RoboDK station: Pick and Place.rdk

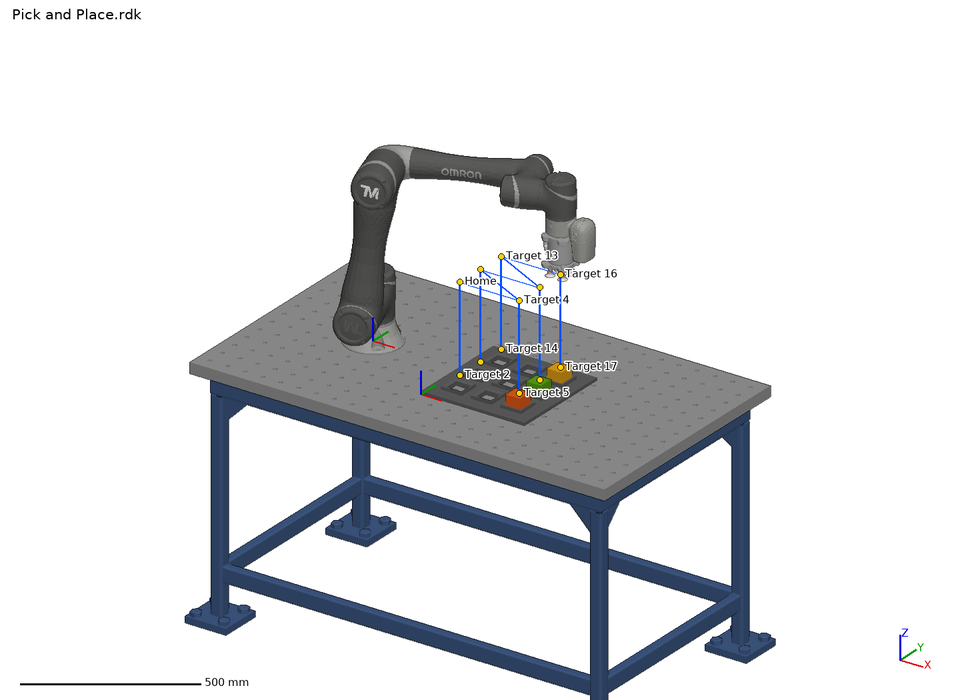
[picture v0: the station drawn from its stored meshes, robots at their saved joint values, targets as dots, program paths as lines]
Station Pick and Place (saved by RoboDK 5.9.2). Poses are relative to the parent item; angles as X-Y-Z fixed-axis rotations.
  - frame Omron TM5-900 Base at (0, 0, 0) mm
    - robot Omron TM5-900: 6 axes, payload 4 kg, reach 900 mm, repeatability 0.05 mm, weight 22.6 kg
        modified DH rows (alpha deg, a mm, theta deg, d mm): 0, 0, 0, 145.2; 90, 0, 90, 0; 0, 429, 0, 0; 0, 411, -90, 122.3; -90, 0, 0, 106.5; 90, 0, 180, 114.15
        joint limits [-270, -180, -155, -180, -180, -270] to [270, 180, 155, 180, 180, 270]; home [0, 0, 90, -90, 90, 0]; saved at [19.778, 6.994, 82.568, 0.438, 90, 19.778]
      - tool SMC ZXP7A01-ZP25C-X1 Vacuum Gripper, TCP at (0, 0, 125) mm, size 88 x 106.8 x 127.9 mm
  - object Table 1400x800x800mm at (0, 0, 0) mm, size 1420 x 820 x 800 mm, geometry from Table-1400x800x800mm.sld
  - frame Reference Frame at (300, -200, 0) mm
    - object Pallete  at (0, 0, 0) mm, size 350 x 350 x 20 mm, geometry from Pallete .step
    - target Home (Cartesian target) at (77.5, 77.7, 335.05) mm, rotated rx 180 ry 0 rz 90 deg; joints [0, -18.954, 105.709, 3.244, 90, 0] of Omron TM5-900
    - target Target 2 (Cartesian target) at (77.5, 77.7, 50) mm, rotated rx 180 ry 0 rz 90 deg; joints [0, -3.452, 137.214, -43.761, 90, 0] of Omron TM5-900
    - target Target 3 (Cartesian target) at (77.5, 77.7, 335) mm, rotated rx 180 ry 0 rz 90 deg; joints [0, -18.954, 105.717, 3.237, 90, 0] of Omron TM5-900
    - target Target 4 (Cartesian target) at (277.5, 77.7, 335) mm, rotated rx 180 ry 0 rz 90 deg; joints [0, 8.043, 81.376, 0.581, 90, 0] of Omron TM5-900
    - target Target 5 (Cartesian target) at (277.5, 77.7, 50) mm, rotated rx 180 ry 0 rz 90 deg; joints [0, 20.58, 108.244, -38.825, 90, 0] of Omron TM5-900
    - target Target 6 (Cartesian target) at (277.5, 77.7, 335) mm, rotated rx 180 ry 0 rz 90 deg; joints [0, 8.043, 81.376, 0.581, 90, 0] of Omron TM5-900
    - target Target 7 (Cartesian target) at (77.5, 177.7, 335) mm, rotated rx 180 ry 0 rz 90 deg; joints [15.489, -21.689, 107.458, 4.231, 90, 15.489] of Omron TM5-900
    - target Target 8 (Cartesian target) at (77.5, 177.7, 50) mm, rotated rx 180 ry 0 rz 90 deg; joints [15.489, -6.322, 139.731, -43.409, 90, 15.489] of Omron TM5-900
    - target Target 9 (Cartesian target) at (77.5, 177.7, 335) mm, rotated rx 180 ry 0 rz 90 deg; joints [15.489, -21.689, 107.458, 4.231, 90, 15.489] of Omron TM5-900
    - target Target 10 (Cartesian target) at (277.5, 177.7, 335) mm, rotated rx 180 ry 0 rz 90 deg; joints [10.006, 6.337, 83.305, 0.358, 90, 10.006] of Omron TM5-900
    - target Target 11 (Cartesian target) at (277.5, 177.7, 50) mm, rotated rx 180 ry 0 rz 90 deg; joints [10.006, 19.191, 110.269, -39.46, 90, 10.006] of Omron TM5-900
    - target Target 12 (Cartesian target) at (277.5, 177.7, 335) mm, rotated rx 180 ry 0 rz 90 deg; joints [10.006, 6.337, 83.305, 0.358, 90, 10.006] of Omron TM5-900
    - target Target 13 (Cartesian target) at (77.5, 277.7, 335) mm, rotated rx 180 ry 0 rz 90 deg; joints [30.132, -20.621, 106.794, 3.828, 90, 30.132] of Omron TM5-900
    - target Target 14 (Cartesian target) at (77.5, 277.7, 50) mm, rotated rx 180 ry 0 rz 90 deg; joints [30.132, -5.185, 138.759, -43.573, 90, 30.132] of Omron TM5-900
    - target Target 15 (Cartesian target) at (77.5, 277.7, 335) mm, rotated rx 180 ry 0 rz 90 deg; joints [30.132, -20.621, 106.794, 3.828, 90, 30.132] of Omron TM5-900
    - target Target 16 (Cartesian target) at (277.5, 277.7, 335) mm, rotated rx 180 ry 0 rz 90 deg; joints [19.778, 6.994, 82.568, 0.438, 90, 19.778] of Omron TM5-900
    - target Target 17 (Cartesian target) at (277.5, 277.7, 50) mm, rotated rx 180 ry 0 rz 90 deg; joints [19.778, 19.728, 109.491, -39.219, 90, 19.778] of Omron TM5-900
    - target Target 18 (Cartesian target) at (277.5, 277.7, 335) mm, rotated rx 180 ry 0 rz 90 deg; joints [19.778, 6.994, 82.568, 0.438, 90, 19.778] of Omron TM5-900
  - program Prog1 (26 instructions, listed below)
  - object Cube 1 at (550, -150, 0) mm, size 50 x 50 x 50 mm, geometry from Cube-50mm.sld
  - object Cube 2 at (500, -200, 0) mm, size 50 x 50 x 50 mm, geometry from Cube-50mm.sld
  - object Cube 3 at (500, -200, 0) mm, size 50 x 50 x 50 mm, geometry from Cube-50mm.sld
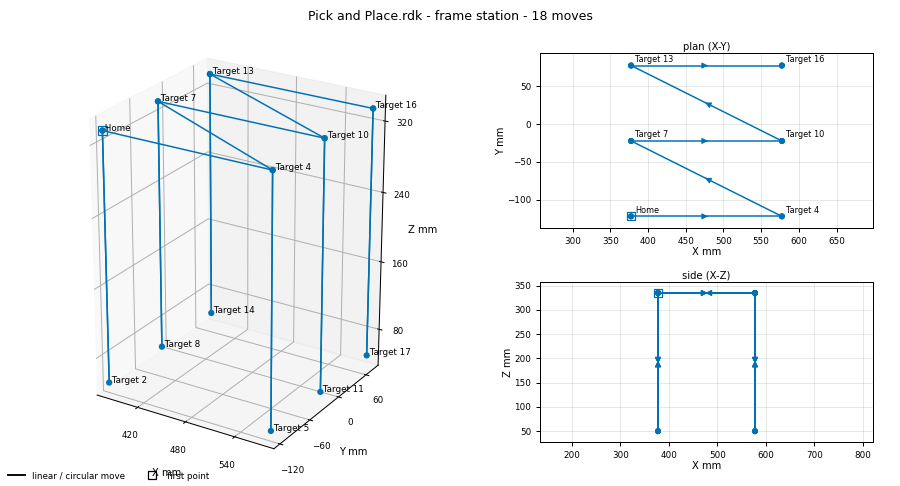
[picture p0: tool path of Pick and Place.rdk in frame station, 18 of 18 moves have a stored position in this frame; points joined in program order, loops and branches not executed]

--- program Prog1 (robot Omron TM5-900) ---
  Set Ref.: Reference Frame
  Set Tool: SMC ZXP7A01-ZP25C-X1 Vacuum Gripper
  MoveL (Home)
  MoveL (Target 2)
  Attach to SMC ZXP7A01-ZP25C-X1 Vacuum Gripper
  MoveL (Target 3)
  MoveL (Target 4)
  MoveL (Target 5)
  Detach from SMC ZXP7A01-ZP25C-X1 Vacuum Gripper
  MoveL (Target 6)
  MoveL (Target 7)
  MoveL (Target 8)
  Attach to SMC ZXP7A01-ZP25C-X1 Vacuum Gripper
  MoveL (Target 9)
  MoveL (Target 10)
  MoveL (Target 11)
  Detach from SMC ZXP7A01-ZP25C-X1 Vacuum Gripper
  MoveL (Target 12)
  MoveL (Target 13)
  MoveL (Target 14)
  Attach to SMC ZXP7A01-ZP25C-X1 Vacuum Gripper
  MoveL (Target 15)
  MoveL (Target 16)
  MoveL (Target 17)
  Detach from SMC ZXP7A01-ZP25C-X1 Vacuum Gripper
  MoveL (Target 18)
